# EPICS alarm handler configuration: mps_database/bareTest/alarms/areas/mpln_l2b_mp03.alhConfig
GROUP NULL MPLN:L2B:MP03:1
$ALIAS MPS Link Node 63
$GUIDANCE
LTUH MPS
   Group Name: MPLN:L2B:MP03:1
   Summary PV:  MPLN:L2B:MP03:1:STATSUMY
$END
CHANNEL  MPLN:L2B:MP03:1    MPLN:L2B:MP03:1:MPS_EN_RBV		-----
CHANNEL  MPLN:L2B:MP03:1    MPLN:L2B:MP03:1:LC1_MODE_RBV		-----
